ABB RobotStudio station: GlueStation_20221110-135028.rsstn

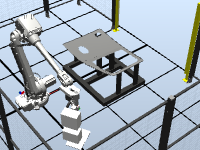
Station GlueStation (saved by RobotStudio 6.8.8307.1040)
Controller IRB4600_20_GlueSystem
  mechanical unit ROB_1: IRB4600_20_250_C_01, 6 joints, base frame (0, 0, 0) mm
Layout (positions relative to the parent item):
  - docking_station [part] at (0, -1345.92, 10) mm, rotated rx 0 ry 0 rz -150 deg
  - SingleDoser [mechanism, from Libraries\SingleDoser.rslib] at (65.32, -1061.16, 1124.58) mm, rotated rx -176.8 ry -12.2 rz 101.89 deg
  - fixture and workpiece [graphiccomponentgroup]
    - door [part]
    - fixture [part]
  - SC_FenceCreator [smart component] at (-1200, -3000, 10) mm
      properties: LengthXside1=4000; LengthXside2=4000; LengthYside1=5300; LengthYside2minus=1500; LengthYside2plus=1500
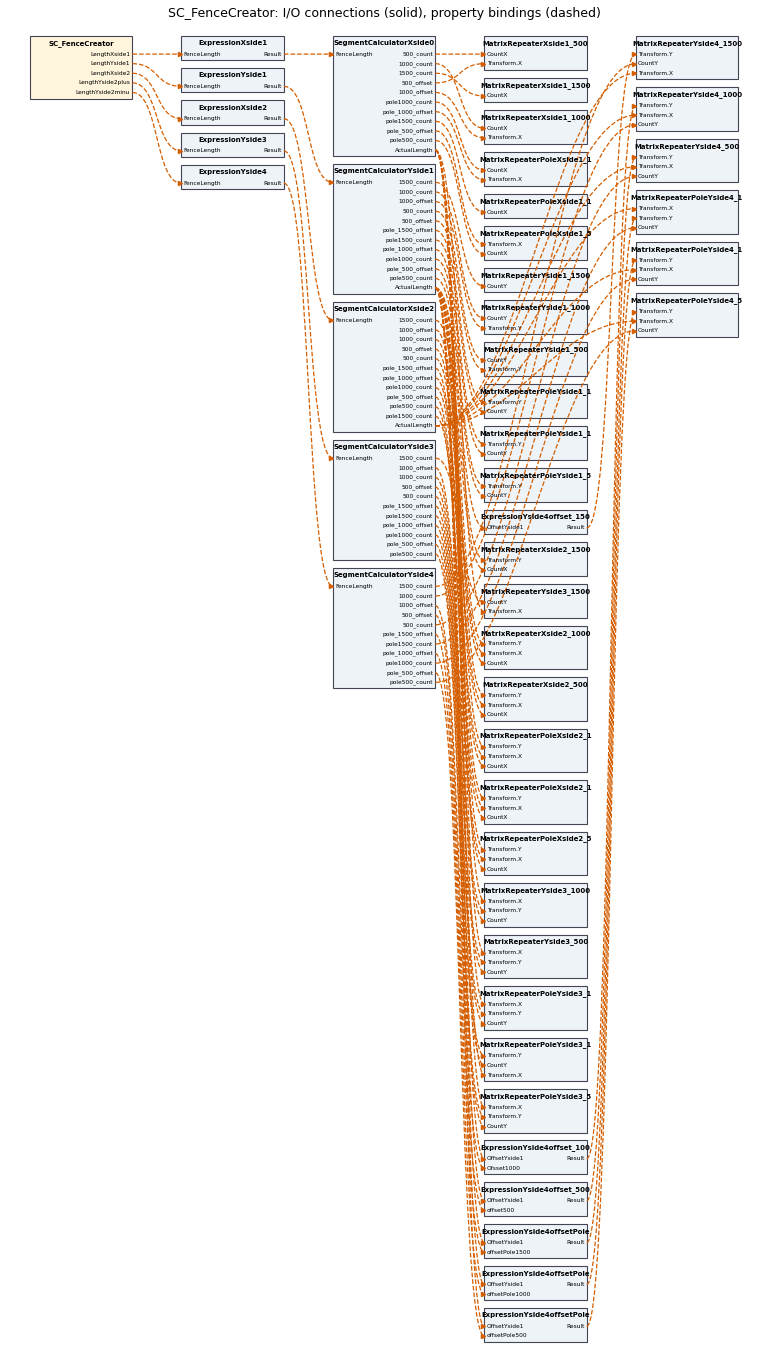
      connections:
        SegmentCalculatorXside0.500_count => MatrixRepeaterXside1_500.CountX
        SegmentCalculatorXside0.1000_count => MatrixRepeaterXside1_1000.CountX
        SegmentCalculatorXside0.1500_count => MatrixRepeaterXside1_1500.CountX
        SegmentCalculatorXside0.500_offset => MatrixRepeaterXside1_500.Transform.X
        SegmentCalculatorXside0.1000_offset => MatrixRepeaterXside1_1000.Transform.X
        SegmentCalculatorXside0.pole1000_count => MatrixRepeaterPoleXside1_1000.CountX
        SegmentCalculatorXside0.pole_1000_offset => MatrixRepeaterPoleXside1_1000.Transform.X
        SegmentCalculatorXside0.pole1500_count => MatrixRepeaterPoleXside1_1500.CountX
        SegmentCalculatorXside0.pole_500_offset => MatrixRepeaterPoleXside1_500.Transform.X
        SegmentCalculatorXside0.pole500_count => MatrixRepeaterPoleXside1_500.CountX
        ExpressionYside1.Result => SegmentCalculatorYside1.FenceLength
        SegmentCalculatorYside1.1500_count => MatrixRepeaterYside1_1500.CountY
        SegmentCalculatorYside1.1000_count => MatrixRepeaterYside1_1000.CountY
        SegmentCalculatorYside1.1000_offset => MatrixRepeaterYside1_1000.Transform.Y
        SegmentCalculatorYside1.500_count => MatrixRepeaterYside1_500.CountY
        SegmentCalculatorYside1.500_offset => MatrixRepeaterYside1_500.Transform.Y
        SegmentCalculatorYside1.pole_1500_offset => MatrixRepeaterPoleYside1_1500.Transform.Y
        SegmentCalculatorYside1.pole1500_count => MatrixRepeaterPoleYside1_1500.CountY
        SegmentCalculatorYside1.pole_1000_offset => MatrixRepeaterPoleYside1_1000.Transform.Y
        SegmentCalculatorYside1.pole1000_count => MatrixRepeaterPoleYside1_1000.CountY
        SegmentCalculatorYside1.pole_500_offset => MatrixRepeaterPoleYside1_500.Transform.Y
        SegmentCalculatorYside1.pole500_count => MatrixRepeaterPoleYside1_500.CountY
        SC_FenceCreator.LengthXside1 => ExpressionXside1.FenceLength
        ExpressionXside2.Result => SegmentCalculatorXside2.FenceLength
        SegmentCalculatorYside1.ActualLength => MatrixRepeaterXside2_1500.Transform.Y
        SegmentCalculatorXside2.1500_count => MatrixRepeaterXside2_1500.CountX
        SegmentCalculatorYside1.ActualLength => MatrixRepeaterXside2_1000.Transform.Y
        SegmentCalculatorXside2.1000_offset => MatrixRepeaterXside2_1000.Transform.X
        SegmentCalculatorXside2.1000_count => MatrixRepeaterXside2_1000.CountX
        SegmentCalculatorYside1.ActualLength => MatrixRepeaterXside2_500.Transform.Y
        SegmentCalculatorXside2.500_offset => MatrixRepeaterXside2_500.Transform.X
        SegmentCalculatorXside2.500_count => MatrixRepeaterXside2_500.CountX
        SegmentCalculatorYside1.ActualLength => MatrixRepeaterPoleXside2_1500.Transform.Y
        SegmentCalculatorXside2.pole_1500_offset => MatrixRepeaterPoleXside2_1500.Transform.X
        SegmentCalculatorYside1.ActualLength => MatrixRepeaterPoleXside2_1000.Transform.Y
        SegmentCalculatorXside2.pole_1000_offset => MatrixRepeaterPoleXside2_1000.Transform.X
        SegmentCalculatorXside2.pole1000_count => MatrixRepeaterPoleXside2_1000.CountX
        SegmentCalculatorYside1.ActualLength => MatrixRepeaterPoleXside2_500.Transform.Y
        SegmentCalculatorXside2.pole_500_offset => MatrixRepeaterPoleXside2_500.Transform.X
        SegmentCalculatorXside2.pole500_count => MatrixRepeaterPoleXside2_500.CountX
        SegmentCalculatorXside2.pole1500_count => MatrixRepeaterPoleXside2_1500.CountX
        SegmentCalculatorYside3.1500_count => MatrixRepeaterYside3_1500.CountY
        ExpressionYside3.Result => SegmentCalculatorYside3.FenceLength
        SegmentCalculatorXside0.ActualLength => MatrixRepeaterYside3_1500.Transform.X
        SegmentCalculatorXside0.ActualLength => MatrixRepeaterYside3_1000.Transform.X
        SegmentCalculatorYside3.1000_offset => MatrixRepeaterYside3_1000.Transform.Y
        SegmentCalculatorYside3.1000_count => MatrixRepeaterYside3_1000.CountY
        SegmentCalculatorXside0.ActualLength => MatrixRepeaterYside3_500.Transform.X
        SegmentCalculatorYside3.500_offset => MatrixRepeaterYside3_500.Transform.Y
        SegmentCalculatorYside3.500_count => MatrixRepeaterYside3_500.CountY
        SegmentCalculatorXside0.ActualLength => MatrixRepeaterPoleYside3_1500.Transform.X
        SegmentCalculatorYside3.pole_1500_offset => MatrixRepeaterPoleYside3_1500.Transform.Y
        SegmentCalculatorYside3.pole1500_count => MatrixRepeaterPoleYside3_1500.CountY
        SegmentCalculatorYside3.pole_1000_offset => MatrixRepeaterPoleYside3_1000.Transform.Y
        SegmentCalculatorYside3.pole1000_count => MatrixRepeaterPoleYside3_1000.CountY
        SegmentCalculatorXside0.ActualLength => MatrixRepeaterPoleYside3_500.Transform.X
        SegmentCalculatorYside3.pole_500_offset => MatrixRepeaterPoleYside3_500.Transform.Y
        SegmentCalculatorYside3.pole500_count => MatrixRepeaterPoleYside3_500.CountY
        SegmentCalculatorXside0.ActualLength => MatrixRepeaterPoleYside3_1000.Transform.X
        ExpressionXside1.Result => SegmentCalculatorXside0.FenceLength
        SC_FenceCreator.LengthYside1 => ExpressionYside1.FenceLength
        SC_FenceCreator.LengthXside2 => ExpressionXside2.FenceLength
        SC_FenceCreator.LengthYside2plus => ExpressionYside3.FenceLength
        SC_FenceCreator.LengthYside2minus => ExpressionYside4.FenceLength
        ExpressionYside4.Result => SegmentCalculatorYside4.FenceLength
        SegmentCalculatorYside1.ActualLength => ExpressionYside4offset_1500.OffsetYside1
        ExpressionYside4offset_1500.Result => MatrixRepeaterYside4_1500.Transform.Y
        SegmentCalculatorYside4.1500_count => MatrixRepeaterYside4_1500.CountY
        SegmentCalculatorXside2.ActualLength => MatrixRepeaterYside4_1500.Transform.X
        SegmentCalculatorYside1.ActualLength => ExpressionYside4offset_1000.OffsetYside1
        ExpressionYside4offset_1000.Result => MatrixRepeaterYside4_1000.Transform.Y
        SegmentCalculatorXside2.ActualLength => MatrixRepeaterYside4_1000.Transform.X
        SegmentCalculatorYside4.1000_count => MatrixRepeaterYside4_1000.CountY
        SegmentCalculatorYside4.1000_offset => ExpressionYside4offset_1000.Ofsset1000
        SegmentCalculatorYside1.ActualLength => ExpressionYside4offset_500.OffsetYside1
        SegmentCalculatorYside4.500_offset => ExpressionYside4offset_500.offset500
        ExpressionYside4offset_500.Result => MatrixRepeaterYside4_500.Transform.Y
        SegmentCalculatorXside2.ActualLength => MatrixRepeaterYside4_500.Transform.X
        SegmentCalculatorYside4.500_count => MatrixRepeaterYside4_500.CountY
        SegmentCalculatorXside2.ActualLength => MatrixRepeaterPoleYside4_1500.Transform.X
        SegmentCalculatorYside1.ActualLength => ExpressionYside4offsetPole_1500.OffsetYside1
        SegmentCalculatorYside4.pole_1500_offset => ExpressionYside4offsetPole_1500.offsetPole1500
        ExpressionYside4offsetPole_1500.Result => MatrixRepeaterPoleYside4_1500.Transform.Y
        SegmentCalculatorYside4.pole1500_count => MatrixRepeaterPoleYside4_1500.CountY
        SegmentCalculatorYside1.ActualLength => ExpressionYside4offsetPole_1000.OffsetYside1
        SegmentCalculatorYside4.pole_1000_offset => ExpressionYside4offsetPole_1000.offsetPole1000
        ExpressionYside4offsetPole_1000.Result => MatrixRepeaterPoleYside4_1000.Transform.Y
        SegmentCalculatorXside2.ActualLength => MatrixRepeaterPoleYside4_1000.Transform.X
        SegmentCalculatorYside4.pole1000_count => MatrixRepeaterPoleYside4_1000.CountY
        SegmentCalculatorYside1.ActualLength => ExpressionYside4offsetPole_500.OffsetYside1
        SegmentCalculatorYside4.pole_500_offset => ExpressionYside4offsetPole_500.offsetPole500
        ExpressionYside4offsetPole_500.Result => MatrixRepeaterPoleYside4_500.Transform.Y
        SegmentCalculatorXside2.ActualLength => MatrixRepeaterPoleYside4_500.Transform.X
        SegmentCalculatorYside4.pole500_count => MatrixRepeaterPoleYside4_500.CountY
    - ExpressionXside1 [smart component, from Libraries\Expression.rslib]
        properties: Expression=FenceLength/1000; FenceLength=4000; Result=4
    - MatrixRepeaterXside1_1500 [smart component, from Libraries\MatrixRepeater.rslib]
        properties: CountX=2; CountY=1; CountZ=1; OffsetX=1.5; OffsetY=0; OffsetZ=0; Source=Panel 2000x1500 X
      - Panel 2000x1500 X [part]
      - Panel 2000x1500 X [part] at (1500, 0, 0) mm
    - MatrixRepeaterXside1_1000 [smart component, from Libraries\MatrixRepeater.rslib] at (3000, 0, 0) mm
        properties: CountX=1; CountY=1; CountZ=1; OffsetX=1; OffsetY=0; OffsetZ=0; Source=Panel 2000x1000 X
      - Panel 2000x1000 X [part]
    - MatrixRepeaterXside1_500 [smart component, from Libraries\MatrixRepeater.rslib] at (4000, 0, 0) mm
        properties: CountX=0; CountY=1; CountZ=1; OffsetX=0.5; OffsetY=0; OffsetZ=0; Source=Panel 2000x500 X
    - MatrixRepeaterPoleXside1_1000 [smart component, from Libraries\MatrixRepeater.rslib] at (4000, 0, 0) mm
        properties: CountX=1; CountY=1; CountZ=1; OffsetX=1; OffsetY=0; OffsetZ=0; Source=Pole
      - Pole [part]
    - Pole [part] at (0, 0, 0) mm
    - SegmentCalculatorXside0 [smart component]
        properties: 1000_count=1; 1000_offset=3; 1500_count=2; 500_count=0; 500_offset=4; ActualLength=4; FenceLength=4; pole_1000_offset=4; pole_1500_offset=0; pole_500_offset=4.5; pole1000_count=1; pole1500_count=3; pole500_count=0; SideNo=0
    - MatrixRepeaterPoleXside1_1500 [smart component, from Libraries\MatrixRepeater.rslib]
        properties: CountX=3; CountY=1; CountZ=1; OffsetX=1.5; OffsetY=0; OffsetZ=1; Source=Pole
      - Pole [part]
      - Pole [part] at (1500, 0, 0) mm
      - Pole [part] at (3000, 0, 0) mm
    - MatrixRepeaterPoleXside1_500 [smart component, from Libraries\MatrixRepeater.rslib] at (4500, 0, 0) mm
        properties: CountX=0; CountY=1; CountZ=1; OffsetX=0.5; OffsetY=0; OffsetZ=0; Source=Pole
    - ExpressionYside1 [smart component, from Libraries\Expression.rslib]
        properties: Expression=FenceLength/1000; FenceLength=5300; Result=5.3
    - MatrixRepeaterYside1_1500 [smart component, from Libraries\MatrixRepeater.rslib]
        properties: CountX=1; CountY=3; CountZ=1; OffsetX=0; OffsetY=1.5; OffsetZ=0; Source=Panel 2000x1500 Y
      - Panel 2000x1500 Y [part]
      - Panel 2000x1500 Y [part] at (0, 1500, 0) mm
      - Panel 2000x1500 Y [part] at (0, 3000, 0) mm
    - MatrixRepeaterYside1_1000 [smart component, from Libraries\MatrixRepeater.rslib] at (0, 4500, 0) mm
        properties: CountX=1; CountY=1; CountZ=1; OffsetX=0; OffsetY=1; OffsetZ=0; Source=Panel 2000x1000 Y
      - Panel 2000x1000 Y [part]
    - MatrixRepeaterYside1_500 [smart component, from Libraries\MatrixRepeater.rslib] at (0, 5500, 0) mm
        properties: CountX=1; CountY=0; CountZ=1; OffsetX=0; OffsetY=0.5; OffsetZ=0; Source=Panel 2000x500 Y
    - PoleYside1 [part] at (0, 0, 0) mm
    - MatrixRepeaterPoleYside1_1500 [smart component, from Libraries\MatrixRepeater.rslib] at (0, 1500, 0) mm
        properties: CountX=1; CountY=3; CountZ=1; OffsetX=0; OffsetY=1.5; OffsetZ=0; Source=PoleYside1
      - PoleYside1 [part]
      - PoleYside1 [part] at (0, 1500, 0) mm
      - PoleYside1 [part] at (0, 3000, 0) mm
    - SegmentCalculatorYside1 [smart component]
        properties: 1000_count=1; 1000_offset=4.5; 1500_count=3; 500_count=0; 500_offset=5.5; ActualLength=5.5; FenceLength=5.3; pole_1000_offset=5.5; pole_1500_offset=1.5; pole_500_offset=6; pole1000_count=1; pole1500_count=3; pole500_count=0; SideNo=1
    - MatrixRepeaterPoleYside1_1000 [smart component, from Libraries\MatrixRepeater.rslib] at (0, 5500, 0) mm
        properties: CountX=1; CountY=1; CountZ=1; OffsetX=0; OffsetY=1; OffsetZ=0; Source=PoleYside1
      - PoleYside1 [part]
    - MatrixRepeaterPoleYside1_500 [smart component, from Libraries\MatrixRepeater.rslib] at (0, 6000, 0) mm
        properties: CountX=1; CountY=0; CountZ=1; OffsetX=0; OffsetY=0.5; OffsetZ=0; Source=PoleYside1
    - PoleXside2 [part] at (0, 0, 0) mm
    - PoleYside3 [part] at (0, 0, 0) mm
    - ExpressionXside2 [smart component, from Libraries\Expression.rslib]
        properties: Expression=FenceLength/1000; FenceLength=4000; Result=4
    - SegmentCalculatorXside2 [smart component]
        properties: 1000_count=1; 1000_offset=3; 1500_count=2; 500_count=0; 500_offset=4; ActualLength=4; FenceLength=4; pole_1000_offset=4; pole_1500_offset=1.5; pole_500_offset=4.5; pole1000_count=1; pole1500_count=2; pole500_count=0; SideNo=2
    - MatrixRepeaterXside2_1500 [smart component, from Libraries\MatrixRepeater.rslib] at (0, 5500, 0) mm
        properties: CountX=2; CountY=1; CountZ=1; OffsetX=1.5; OffsetY=0; OffsetZ=0; Source=Panel 2000x1500 X
      - Panel 2000x1500 X [part]
      - Panel 2000x1500 X [part] at (1500, 0, 0) mm
    - MatrixRepeaterXside2_1000 [smart component, from Libraries\MatrixRepeater.rslib] at (3000, 5500, 0) mm
        properties: CountX=1; CountY=1; CountZ=1; OffsetX=1; OffsetY=0; OffsetZ=0; Source=Panel 2000x1000 X
      - Panel 2000x1000 X [part]
    - MatrixRepeaterXside2_500 [smart component, from Libraries\MatrixRepeater.rslib] at (4000, 5500, 0) mm
        properties: CountX=0; CountY=1; CountZ=1; OffsetX=0.5; OffsetY=0; OffsetZ=0; Source=Panel 2000x500 X
    - MatrixRepeaterPoleXside2_1500 [smart component, from Libraries\MatrixRepeater.rslib] at (1500, 5500, 0) mm
        properties: CountX=2; CountY=1; CountZ=1; OffsetX=1.5; OffsetY=0; OffsetZ=0; Source=PoleXside2
      - PoleXside2 [part]
      - PoleXside2 [part] at (1500, 0, 0) mm
    - MatrixRepeaterPoleXside2_1000 [smart component, from Libraries\MatrixRepeater.rslib] at (4000, 5500, 0) mm
        properties: CountX=1; CountY=1; CountZ=1; OffsetX=1; OffsetY=0; OffsetZ=0; Source=PoleXside2
      - PoleXside2 [part]
    - MatrixRepeaterPoleXside2_500 [smart component, from Libraries\MatrixRepeater.rslib] at (4500, 5500, 0) mm
        properties: CountX=0; CountY=1; CountZ=1; OffsetX=0.5; OffsetY=0; OffsetZ=0; Source=PoleXside2
    - SegmentCalculatorYside3 [smart component]
        properties: 1000_count=0; 1000_offset=1.5; 1500_count=1; 500_count=0; 500_offset=1.5; ActualLength=1.5; FenceLength=1.5; pole_1000_offset=2.5; pole_1500_offset=1.5; pole_500_offset=2; pole1000_count=0; pole1500_count=1; pole500_count=0; SideNo=3
    - ExpressionYside3 [smart component]
        properties: Expression=FenceLength/1000; FenceLength=1500; Result=1.5
    - MatrixRepeaterYside3_1500 [smart component] at (4000, 0, 0) mm
        properties: CountX=1; CountY=1; CountZ=1; OffsetX=0; OffsetY=1.5; OffsetZ=0; Source=Panel 2000x1500 Y
      - Panel 2000x1500 Y [part]
    - MatrixRepeaterYside3_1000 [smart component] at (4000, 1500, 0) mm
        properties: CountX=1; CountY=0; CountZ=1; OffsetX=0; OffsetY=1; OffsetZ=0; Source=Panel 2000x1000 Y
    - MatrixRepeaterYside3_500 [smart component] at (4000, 1500, 0) mm
        properties: CountX=1; CountY=0; CountZ=1; OffsetX=0; OffsetY=0.5; OffsetZ=0; Source=Panel 2000x500 Y
    - MatrixRepeaterPoleYside3_1500 [smart component] at (4000, 1500, 0) mm
        properties: CountX=1; CountY=1; CountZ=1; OffsetX=0; OffsetY=1.5; OffsetZ=0; Source=PoleYside3
      - PoleYside3 [part]
    - MatrixRepeaterPoleYside3_1000 [smart component] at (4000, 2500, 0) mm
        properties: CountX=1; CountY=0; CountZ=1; OffsetX=0; OffsetY=1; OffsetZ=0; Source=PoleYside3
    - MatrixRepeaterPoleYside3_500 [smart component] at (4000, 2000, 0) mm
        properties: CountX=1; CountY=0; CountZ=1; OffsetX=0; OffsetY=0.5; OffsetZ=0; Source=PoleYside3
    - ExpressionYside4 [smart component, from Libraries\Expression.rslib]
        properties: Expression=FenceLength/1000; FenceLength=1500; Result=1.5
    - SegmentCalculatorYside4 [smart component]
        properties: 1000_count=0; 1000_offset=1.5; 1500_count=1; 500_count=0; 500_offset=1.5; ActualLength=1.5; FenceLength=1.5; pole_1000_offset=2.5; pole_1500_offset=1.5; pole_500_offset=2; pole1000_count=0; pole1500_count=1; pole500_count=0; SideNo=4
    - MatrixRepeaterYside4_1500 [smart component, from Libraries\MatrixRepeater.rslib] at (4000, 4000, 0) mm
        properties: CountX=1; CountY=1; CountZ=1; OffsetX=0; OffsetY=-1.5; OffsetZ=0; Source=Panel 2000x1500 Y
      - Panel 2000x1500 Y [part]
    - ExpressionYside4offset_1500 [smart component, from Libraries\Expression.rslib]
        properties: Expression=OffsetYside1-1.5; OffsetYside1=5.5; Result=4
    - ExpressionYside4offset_1000 [smart component, from Libraries\Expression.rslib]
        properties: Expression=OffsetYside1-Ofsset1000-1; OffsetYside1=5.5; Ofsset1000=1.5; Result=3
    - MatrixRepeaterYside4_1000 [smart component, from Libraries\MatrixRepeater.rslib] at (4000, 3000, 0) mm
        properties: CountX=1; CountY=0; CountZ=1; OffsetX=0; OffsetY=-1; OffsetZ=0; Source=Panel 2000x1000 Y
    - ExpressionYside4offset_500 [smart component, from Libraries\Expression.rslib]
        properties: Expression=OffsetYside1-offset500-0.5; offset500=1.5; OffsetYside1=5.5; Result=3.5
    - MatrixRepeaterYside4_500 [smart component, from Libraries\MatrixRepeater.rslib] at (4000, 3500, 0) mm
        properties: CountX=1; CountY=0; CountZ=1; OffsetX=0; OffsetY=-0.5; OffsetZ=0; Source=Panel 2000x500 Y
    - MatrixRepeaterPoleYside4_1500 [smart component, from Libraries\MatrixRepeater.rslib] at (4000, 4000, 0) mm
        properties: CountX=1; CountY=1; CountZ=1; OffsetX=0; OffsetY=-1.5; OffsetZ=0; Source=PoleYside3
      - PoleYside3 [part]
    - ExpressionYside4offsetPole_1500 [smart component, from Libraries\Expression.rslib]
        properties: Expression=OffsetYside1-offsetPole1500; offsetPole1500=1.5; OffsetYside1=5.5; Result=4
    - ExpressionYside4offsetPole_1000 [smart component, from Libraries\Expression.rslib]
        properties: Expression=OffsetYside1-offsetPole1000; offsetPole1000=2.5; OffsetYside1=5.5; Result=3
    - MatrixRepeaterPoleYside4_1000 [smart component, from Libraries\MatrixRepeater.rslib] at (4000, 3000, 0) mm
        properties: CountX=1; CountY=0; CountZ=1; OffsetX=0; OffsetY=-1; OffsetZ=0; Source=PoleYside3
    - ExpressionYside4offsetPole_500 [smart component, from Libraries\Expression.rslib]
        properties: Expression=OffsetYside1-offsetPole500; offsetPole500=2; OffsetYside1=5.5; Result=3.5
    - MatrixRepeaterPoleYside4_500 [smart component, from Libraries\MatrixRepeater.rslib] at (4000, 3500, 0) mm
        properties: CountX=1; CountY=0; CountZ=1; OffsetX=0; OffsetY=-0.5; OffsetZ=0; Source=PoleYside3
    - Panel 2000x1000 X [part]
    - Panel 2000x1500 X [part]
    - Panel 2000x500 X [part]
    - Panel 2000x1000 Y [part]
    - Panel 2000x1500 Y [part]
    - Panel 2000x500 Y [part]
  - SC_LightGuard [smart component] at (2800, -1416, 10) mm, rotated rx 0 ry 0 rz 90 deg
      properties: GuardDistance=2330; vecPosition=[0 0 0]; vecOrientation=[0 0 0]
      signals: DI UpdateDistance, DI diGuardOn
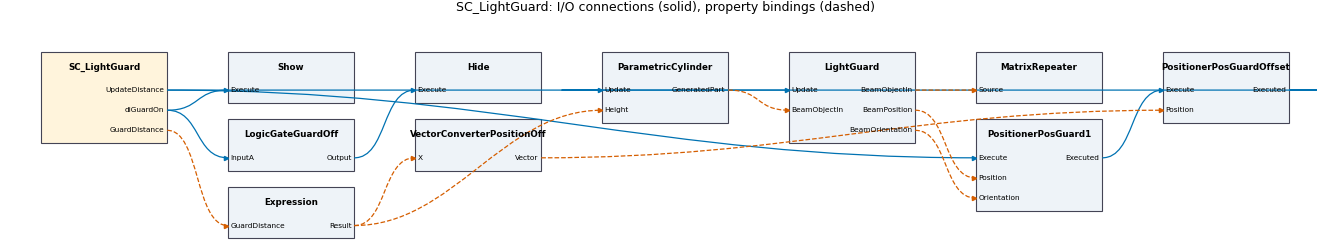
      connections:
        SC_LightGuard.UpdateDistance -> LightGuard.Update
        SC_LightGuard.UpdateDistance -> PositionerPosGuard1.Execute
        PositionerPosGuard1.Executed -> PositionerPosGuardOffset.Execute
        PositionerPosGuardOffset.Executed -> ParametricCylinder.Update
        SC_LightGuard.diGuardOn -> Show.Execute
        SC_LightGuard.diGuardOn -> LogicGateGuardOff.InputA
        LogicGateGuardOff.Output -> Hide.Execute
        SC_LightGuard.GuardDistance => Expression.GuardDistance
        Expression.Result => VectorConverterPositionOffset.X
        VectorConverterPositionOffset.Vector => PositionerPosGuardOffset.Position
        Expression.Result => ParametricCylinder.Height
        ParametricCylinder.GeneratedPart => LightGuard.BeamObjectIn
        LightGuard.BeamObjectIn => MatrixRepeater.Source
        LightGuard.BeamPosition => PositionerPosGuard1.Position
        LightGuard.BeamOrientation => PositionerPosGuard1.Orientation
    - light_guard2 [part] at (2330, 0, 0) mm
    - light_guard1 [part]
    - PositionerPosGuard1 [smart component]
        properties: Object=light_guard2; Position=[2.8 -1.416 0.01]; Orientation=[0 0 1.5707963267949]; Reference=Global; ReferenceObject=SC_LightGuard
        signals: DI Execute, DO Executed
    - Expression [smart component]
        properties: Expression=GuardDistance/1000; Result=2.33; GuardDistance=2330
    - PositionerPosGuardOffset [smart component]
        properties: Object=light_guard2; Position=[2.33 0 0]; Orientation=[0 0 0]; Reference=Local; ReferenceObject=(none)
        signals: DI Execute, DO Executed
    - VectorConverterPositionOffset [smart component]
        properties: X=2.33; Y=0; Z=0; Vector=[2.33 0 0]
    - ParametricCylinder [smart component] at (0, 0, 200) mm, rotated rx 0 ry 90 rz 0 deg
        properties: Radius=0.002; Height=2.33; GeneratedPart=GeneratedPart; KeepGeometry=true
        signals: DI Update
      - GeneratedPart [part]
    - MatrixRepeater [smart component] at (0, 0, 200) mm, rotated rx 0 ry 90 rz 0 deg
        properties: Source=GeneratedPart; CountX=32; CountY=1; CountZ=1; OffsetX=-0.05; OffsetY=0; OffsetZ=0
      - GeneratedPart [part]
      - GeneratedPart [part] at (-50, 0, 0) mm
      - GeneratedPart [part] at (-100, 0, 0) mm
      - GeneratedPart [part] at (-150, 0, 0) mm
      - GeneratedPart [part] at (-200, 0, 0) mm
      - GeneratedPart [part] at (-250, 0, 0) mm
      - GeneratedPart [part] at (-300, 0, 0) mm
      - GeneratedPart [part] at (-350, 0, 0) mm
      - GeneratedPart [part] at (-400, 0, 0) mm
      - GeneratedPart [part] at (-450, 0, 0) mm
      - GeneratedPart [part] at (-500, 0, 0) mm
      - GeneratedPart [part] at (-550, 0, 0) mm
      - GeneratedPart [part] at (-600, 0, 0) mm
      - GeneratedPart [part] at (-650, 0, 0) mm
      - GeneratedPart [part] at (-700, 0, 0) mm
      - GeneratedPart [part] at (-750, 0, 0) mm
      - GeneratedPart [part] at (-800, 0, 0) mm
      - GeneratedPart [part] at (-850, 0, 0) mm
      - GeneratedPart [part] at (-900, 0, 0) mm
      - GeneratedPart [part] at (-950, 0, 0) mm
      - GeneratedPart [part] at (-1000, 0, 0) mm
      - GeneratedPart [part] at (-1050, 0, 0) mm
      - GeneratedPart [part] at (-1100, 0, 0) mm
      - GeneratedPart [part] at (-1150, 0, 0) mm
      - GeneratedPart [part] at (-1200, 0, 0) mm
      - GeneratedPart [part] at (-1250, 0, 0) mm
      - GeneratedPart [part] at (-1300, 0, 0) mm
      - GeneratedPart [part] at (-1350, 0, 0) mm
      - GeneratedPart [part] at (-1400, 0, 0) mm
      - GeneratedPart [part] at (-1450, 0, 0) mm
      - GeneratedPart [part] at (-1500, 0, 0) mm
      - GeneratedPart [part] at (-1550, 0, 0) mm
    - Show [smart component]
        properties: Object=MatrixRepeater
        signals: DI Execute, DO Executed
    - Hide [smart component]
        properties: Object=MatrixRepeater
        signals: DI Execute, DO Executed
    - LogicGateGuardOff [smart component]
        properties: Operator=NOT; Delay=0
        signals: DI InputA, DI InputB, DO Output
    - LightGuard [smart component]
        properties: BeamObjectIn=GeneratedPart; LightGuard=light_guard1; BeamObjectOut=GeneratedPart; BeamPosition=[2.8 -1.416 0.01]; BeamOrientation=[0 0 1.5707963267949]
        signals: DI Update
  - IRB4600_20_250_C_01 [mechanism, from Robots\IRB4600_20_250_C_G_01.rslib] at (0, 0, 0) mm; joint values [-1.5026, -0.2673, 0.6887, -0.0867, 1.3535, -0.1179] (rad or m)
Attachment: SingleDoser is attached to IRB4600_20_250_C_01 / Link6
Targets, tools, work objects and paths stored in the station, written as RAPID:
! task T_ROB1
MODULE modRobotStudio
  CONST robtarget pDockingStn:=[[-6.21722435,13.985562095,-127.5],[0,0.737075919,0.675809951,0],[-1,0,0,0],[9E+09,9E+09,9E+09,9E+09,9E+09,9E+09]];
  CONST robtarget pAboveDockingStn:=[[-6.217297914,13.985583992,22.500016978],[-0.000000026,0.737075879,0.675809995,-0.000000022],[-1,0,0,0],[9E+09,9E+09,9E+09,9E+09,9E+09,9E+09]];
  PROC FromDockingStation()
    MoveJ pDockingStn,v200,z1,tNozzle\WObj:=wobjDockingStn;
    MoveL pAboveDockingStn,v200,z1,tNozzle\WObj:=wobjDockingStn;
  ENDPROC
  PROC ToDockingStation()
    MoveL pAboveDockingStn,v1000,z1,tNozzle\WObj:=wobjDockingStn;
    MoveL pDockingStn,v200,fine,tNozzle\WObj:=wobjDockingStn;
  ENDPROC
ENDMODULE

! task T_ROB1
MODULE modCalibData
  TASK PERS wobjdata wobjDockingStn:=[FALSE,TRUE,"",[[93.58826629,-1285.222736121,827.125],[0.818981032,0,0,-0.57382059]],[[0,0,0],[1,0,0,0]]];
ENDMODULE

! task T_ROB1
MODULE CalibData
  PERS tooldata tNozzle:=[TRUE,[[-305.801192078,0,351.776515421],[0.991444861,0,-0.130526192,0]],[10,[-216.957886762,-4.684934403,103.554004337],[1,0,0,0],0,0,0]];
ENDMODULE

! task T_ROB1
MODULE modCalibData
  PERS tooldata tNozzle:=[TRUE,[[-305.801192078,0,351.776515421],[0.991444861,0,-0.130526192,0]],[10,[-216.957886762,-4.684934403,103.554004337],[1,0,0,0],0,0,0]];
  TASK PERS wobjdata wobjDockingStn:=[FALSE,TRUE,"",[[93.58826629,-1285.222736121,827.125],[0.818981032,0,0,-0.57382059]],[[0,0,0],[1,0,0,0]]];
ENDMODULE

! task T_ROB1
MODULE modRobotStudio
  CONST robtarget pDockingStn:=[[-6.21722435,13.985562095,-127.5],[0,0.737075919,0.675809951,0],[-1,0,0,0],[9E+09,9E+09,9E+09,9E+09,9E+09,9E+09]];
  CONST robtarget pAboveDockingStn:=[[-6.217297914,13.985583992,22.500016978],[-0.000000026,0.737075879,0.675809995,-0.000000022],[-1,0,0,0],[9E+09,9E+09,9E+09,9E+09,9E+09,9E+09]];
  PROC FromDockingStation()
    MoveJ pDockingStn,v200,z1,tNozzle\WObj:=wobjDockingStn;
    MoveL pAboveDockingStn,v200,z1,tNozzle\WObj:=wobjDockingStn;
  ENDPROC
  PROC ToDockingStation()
    MoveL pAboveDockingStn,v1000,z1,tNozzle\WObj:=wobjDockingStn;
    MoveL pDockingStn,v200,fine,tNozzle\WObj:=wobjDockingStn;
  ENDPROC
ENDMODULE

